Staubli VAL3: CircleCenter.dtx

bool bExit
public bool bFrameSave
bool bFrameTeach
bool bOk
bool bSame = true
frame fFrame1 = {fatherId=world[0]}
frame fFrameRef = {fatherId=world[0]}
mdesc mNomSpeed
num nAngle
num nDia
num nFrame1Err = -1
num nItem[6]
num nMax[6]
num nMin[6]
num nSelectedPt = 2
num nStatus = 2
num nWorkingMode = 3
public pointRx pFrameRefPt[3]
  [0] = {x=250, z=1944, shoulder=lefty, elbow=epositive, wrist=wpositive, fatherId=world[0]}
  [1] = {x=250, z=1944, shoulder=lefty, elbow=epositive, wrist=wpositive, fatherId=world[0]}
  [2] = {x=250, z=1944, shoulder=lefty, elbow=epositive, wrist=wpositive, fatherId=world[0]}
pointRx pPointCenter = {fatherId=world[0]}
string sButton[2]
  [0] = "是"
  [1] = "否"
string sCutPosStatus
string sEmptyOrNotC[3]
string sItem[6]
string sOffSet[6]
  [0] = "X:  1460.6 "
  [1] = "Y:  35.71"
  [2] = "Z:  -199.19"
  [3] = "Rx: -0.12"
  [4] = "Ry: -0.31"
  [5] = "Rz: -53.75"
string sThreeOffset[3]
  [0] = "第1点(圆周上)"
  [1] = "第2点(圆周上)"
  [2] = "第3点(圆周上)"
tool tTool = {fatherId=flange[0], ioLink=valve1}
trsf trFrame
trsf trOffSetOut
trsf trOffset
